{attribute 'OPC.UA.DA.StructuredType' := '1'}
TYPE ST_CondensingBoilerState :
STRUCT
	bError					: BOOL;
END_STRUCT
END_TYPE

(* stored: Version 1.1.0.1, ProductVersion 3.1.4024.10
   DUT ST_CondensingBoilerState: Id {f1edab42-1801-4621-844b-038f7355bd8a} *)
